SYSTEM FIO_Sorting_Station
  (* Version 1.0, 2022-03-11, Maximilian Scharf *)
  APPLICATION Sorting_Station
    (* Group __Group01: Human Machine Interface *)
    (* Group __Group02: Sensors *)
    (* Group __Group03: Factory IO data *)
    (* Group __Group04: Aktuatoren *)
    (* Group __Group05: Human Machine Interface *)
    (* Group __Group07: Factory IO data *)
    (* Group __Group09: Counter Ticker *)
    FBS
      E_R_TRIG : E_R_TRIG;
      BOOL2BOOL : BOOL2BOOL; {SET_ATTRIBUTE(GroupName, __Group02)}
      BOOL2BOOL_1 : BOOL2BOOL; {SET_ATTRIBUTE(GroupName, __Group01)}
      BOOL2BOOL_2 : BOOL2BOOL; {SET_ATTRIBUTE(GroupName, __Group01)}
      BOOL2BOOL_3 : BOOL2BOOL; {SET_ATTRIBUTE(GroupName, __Group01)}
      BOOL2BOOL_4 : BOOL2BOOL; {SET_ATTRIBUTE(GroupName, __Group01)}
      BOOL2BOOL_5 : BOOL2BOOL; {SET_ATTRIBUTE(GroupName, __Group01)}
      BOOL2BOOL_6 : BOOL2BOOL; {SET_ATTRIBUTE(GroupName, __Group01)}
      BOOL2BOOL_7 : BOOL2BOOL(IN := 0);
      BOOL2BOOL_8 : BOOL2BOOL(IN := 0);
      BOOL2BOOL_9 : BOOL2BOOL(IN := 0);
      BOOL2BOOL_10 : BOOL2BOOL(IN := 0);
      BOOL2BOOL_11 : BOOL2BOOL(IN := 0);
      BOOL2BOOL_18 : BOOL2BOOL;
      E_R_TRIG_2 : E_R_TRIG;
      Is_running : E_RS;
      E_F_TRIG : E_F_TRIG;
      Is_running_NOT : F_NOT;
      UINT2UINT : F_DINT_TO_UINT; {SET_ATTRIBUTE(GroupName, __Group02)}
      E_R_TRIG_1 : E_R_TRIG;
      F_SEL : F_SEL(IN0 := UINT#1);
      UINT2UINT_1 : UINT2UINT;
      UINT2UINT_2 : UINT2UINT;
      BOOL2BOOL_12 : BOOL2BOOL;
      UINT2UINT_3 : UINT2UINT;
      BOOL2BOOL_13 : BOOL2BOOL;
      UINT2UINT_4 : UINT2UINT;
      BOOL2BOOL_14 : BOOL2BOOL;
      BOOL2BOOL_15 : BOOL2BOOL;
      UINT2UINT_5 : UINT2UINT;
      UINT2UINT_6 : UINT2UINT; {SET_ATTRIBUTE(GroupName, __Group09)}
      BOOL2BOOL_16 : BOOL2BOOL;
      BOOL2BOOL_17 : BOOL2BOOL;
      UINT2UINT_7 : UINT2UINT;
      UINT2UINT_8 : UINT2UINT;
      UINT2UINT_9 : UINT2UINT; {SET_ATTRIBUTE(GroupName, __Group09)}
      UINT2UINT_10 : UINT2UINT; {SET_ATTRIBUTE(GroupName, __Group09)}
      BOOL2BOOL_19 : BOOL2BOOL;
      E_R_TRIG_3 : E_R_TRIG;
      BOOL2BOOL_20 : BOOL2BOOL;
      E_R_TRIG_4 : E_R_TRIG;
      BOOL2BOOL_21 : BOOL2BOOL;
      E_R_TRIG_5 : E_R_TRIG;
    END_FBS
    SUBAPPS
      FIO : OPC_SUB_FIO(QI := 1); {SET_ATTRIBUTE(GroupName, __Group03)}
      UPC_PUB_FIO : OPC_PUB_FIO(QI := 1); {SET_ATTRIBUTE(GroupName, __Group07)}
      Start_Light : OPC_PUB_1_FixID(QI := 1, prefix := "FIO_Q_", var1 := "start_light"); {SET_ATTRIBUTE(GroupName, __Group05)}
      Reset_Light : OPC_PUB_1_FixID(QI := 1, prefix := "FIO_Q_", var1 := "reset_light"); {SET_ATTRIBUTE(GroupName, __Group05)}
      Stop_Light : OPC_PUB_1_FixID(QI := 1, prefix := "FIO_Q_", var1 := "stop_light"); {SET_ATTRIBUTE(GroupName, __Group05)}
      ENTRY_CONVEYOR : OPC_PUB_1_FixID(QI := 1, prefix := "FIO_Q_", var1 := "entry_conveyor"); {SET_ATTRIBUTE(GroupName, __Group04)}
      EXIT_CONVEYOR : OPC_PUB_1_FixID(QI := 1, prefix := "FIO_Q_", var1 := "exit_conveyor"); {SET_ATTRIBUTE(GroupName, __Group04)}
      At_Exit : OPC_SUB_1_FixID(QI := 1, prefix := "FIO_I_", var1 := "at_exit"); {SET_ATTRIBUTE(GroupName, __Group02)}
      Vison_Sensor : OPC_SUB_1_FixID(QI := 1, prefix := "FIO_I_", var1 := "vision_sensor"); {SET_ATTRIBUTE(GroupName, __Group02)}
      Stop : OPC_SUB_1_FixID(QI := 1, prefix := "FIO_I_", var1 := "Stop"); {SET_ATTRIBUTE(GroupName, __Group01)}
      Reset : OPC_SUB_1_FixID(QI := 1, prefix := "FIO_I_", var1 := "reset"); {SET_ATTRIBUTE(GroupName, __Group01)}
      Emergency_Stop : OPC_SUB_1_FixID(QI := 1, prefix := "FIO_I_", var1 := "emergency_stop"); {SET_ATTRIBUTE(GroupName, __Group01)}
      Auto : OPC_SUB_1_FixID(QI := 1, prefix := "FIO_I_", var1 := "auto"); {SET_ATTRIBUTE(GroupName, __Group01)}
      Manual : OPC_SUB_1_FixID(QI := 1, prefix := "FIO_I_", var1 := "Manual"); {SET_ATTRIBUTE(GroupName, __Group01)}
      Start : OPC_SUB_1_FixID(QI := 1, prefix := "FIO_I_", var1 := "start"); {SET_ATTRIBUTE(GroupName, __Group01)}
      STOP_BLADE : OPC_PUB_1_FixID(QI := 1, prefix := "FIO_Q_", var1 := "stop_blade"); {SET_ATTRIBUTE(GroupName, __Group04)}
      Sorter_1 : Sorter(Prefix := "FIO_Q_", CountVar := "counter_1", BeltVar := "sorter_1_belt", TurnVar := "sorter_1_turn"); {SET_ATTRIBUTE(GroupName, __Group04)}
      Sorter_2 : Sorter(Prefix := "FIO_Q_", CountVar := "counter_2", BeltVar := "sorter_2_belt", TurnVar := "sorter_2_turn"); {SET_ATTRIBUTE(GroupName, __Group04)}
      Sorter_3 : Sorter(Prefix := "FIO_Q_", CountVar := "counter_3", BeltVar := "sorter_3_belt", TurnVar := "sorter_3_turn"); {SET_ATTRIBUTE(GroupName, __Group04)}
      OPC_PUB_1_FixID : OPC_PUB_1_FixID(QI := 1, prefix := "CON_", var1 := "sorter_1");
      OPC_PUB_EX_1 : OPC_PUB_EX_1(QI := 1, prefix := "FIO_Q_", var1 := "sorter_1_belt", server := WSTRING#"localhost:4840");
      OPC_PUB_EX_2 : OPC_PUB_EX_1(QI := 1, prefix := "FIO_Q_", var1 := "sorter_1_turn", server := WSTRING#"localhost:4840");
      OPC_SUB_EX_4 : OPC_SUB_EX_1(QI := 1, prefix := "CON_", var1 := "sorter_1", server := WSTRING#"localhost:4840");
      OPC_SUB_EX_5 : OPC_SUB_EX_1(QI := 1, prefix := "CON_", var1 := "sorter_2", server := WSTRING#"localhost:4840");
      OPC_PUB_EX_3 : OPC_PUB_EX_1(QI := 1, prefix := "FIO_Q_", var1 := "sorter_2_belt", server := WSTRING#"localhost:4840");
      OPC_PUB_EX_4 : OPC_PUB_EX_1(QI := 1, prefix := "FIO_Q_", var1 := "sorter_2_turn", server := WSTRING#"localhost:4840");
      OPC_PUB_EX_5 : OPC_PUB_EX_1(QI := 1, prefix := "FIO_Q_", var1 := "sorter_3_belt", server := WSTRING#"localhost:4840");
      OPC_SUB_EX_6 : OPC_SUB_EX_1(QI := 1, prefix := "CON_", var1 := "sorter_3", server := WSTRING#"localhost:4840");
      OPC_PUB_EX_6 : OPC_PUB_EX_1(QI := 1, prefix := "FIO_Q_", var1 := "sorter_3_turn", server := WSTRING#"localhost:4840");
      OPC_PUB_1_FixID_1 : OPC_PUB_1_FixID(QI := 1, prefix := "CON_", var1 := "sorter_2");
      OPC_PUB_1_FixID_2 : OPC_PUB_1_FixID(QI := 1, prefix := "CON_", var1 := "sorter_3");
      SorterLogic : SorterLogic(PackageNum := UINT#1);
      SorterLogic_3 : SorterLogic(PackageNum := UINT#2);
      SorterLogic_1 : SorterLogic(PackageNum := UINT#3);
      OPC_SUB_EX_7 : OPC_SUB_EX_1(QI := 1, prefix := "FIO_I_", var1 := "at_exit", server := WSTRING#"localhost:4840");
      OPC_SUB_1_FixID : OPC_SUB_1_FixID(QI := 1, prefix := "CON_", var1 := "C1"); {SET_ATTRIBUTE(GroupName, __Group09)}
      OPC_PUB_EX_7 : OPC_PUB_EX_1(QI := 1, prefix := "CON_", var1 := "C1", server := WSTRING#"localhost:4840");
      OPC_SUB_EX_8 : OPC_SUB_EX_1(QI := 1, prefix := "FIO_I_", var1 := "at_exit", server := WSTRING#"localhost:4840");
      OPC_SUB_EX_9 : OPC_SUB_EX_1(QI := 1, prefix := "FIO_I_", var1 := "at_exit", server := WSTRING#"localhost:4840");
      OPC_PUB_EX_8 : OPC_PUB_EX_1(QI := 1, prefix := "CON_", var1 := "C2", server := WSTRING#"localhost:4840");
      OPC_PUB_EX_9 : OPC_PUB_EX_1(QI := 1, prefix := "CON_", var1 := "C3", server := WSTRING#"localhost:4840");
      OPC_SUB_1_FixID_1 : OPC_SUB_1_FixID(QI := 1, prefix := "CON_", var1 := "C2"); {SET_ATTRIBUTE(GroupName, __Group09)}
      OPC_SUB_1_FixID_2 : OPC_SUB_1_FixID(QI := 1, prefix := "CON_", var1 := "C3"); {SET_ATTRIBUTE(GroupName, __Group09)}
      OPC_SUB_EX_1 : OPC_SUB_EX_1(QI := 1, prefix := "FIO_I_", var1 := "reset", server := WSTRING#"localhost:4840");
      OPC_SUB_EX_2 : OPC_SUB_EX_1(QI := 1, prefix := "FIO_I_", var1 := "reset", server := WSTRING#"localhost:4840");
      OPC_SUB_EX_3 : OPC_SUB_EX_1(QI := 1, prefix := "FIO_I_", var1 := "reset", server := WSTRING#"localhost:4840");
    END_SUBAPPS
    EVENT_CONNECTIONS
      BOOL2BOOL.CNF TO E_R_TRIG.EI;
      FIO.INITO TO UPC_PUB_FIO.INIT;
      At_Exit.IND TO BOOL2BOOL.REQ;
      Reset.IND TO BOOL2BOOL_1.REQ;
      Stop.IND TO BOOL2BOOL_3.REQ;
      Emergency_Stop.IND TO BOOL2BOOL_4.REQ;
      Auto.IND TO BOOL2BOOL_5.REQ;
      Manual.IND TO BOOL2BOOL_6.REQ;
      BOOL2BOOL_7.CNF TO Start_Light.REQ;
      BOOL2BOOL_8.CNF TO Reset_Light.REQ;
      BOOL2BOOL_9.CNF TO Stop_Light.REQ;
      BOOL2BOOL_10.CNF TO ENTRY_CONVEYOR.REQ;
      BOOL2BOOL_11.CNF TO EXIT_CONVEYOR.REQ;
      Start.IND TO BOOL2BOOL_2.REQ;
      BOOL2BOOL_18.CNF TO STOP_BLADE.REQ;
      BOOL2BOOL_2.CNF TO E_R_TRIG_2.EI;
      E_R_TRIG_2.EO TO Is_running.S;
      Is_running.EO TO BOOL2BOOL_7.REQ;
      Is_running.EO TO BOOL2BOOL_10.REQ;
      Is_running.EO TO BOOL2BOOL_11.REQ;
      BOOL2BOOL_3.CNF TO E_F_TRIG.EI;
      E_F_TRIG.EO TO Is_running.R;
      Is_running.EO TO Is_running_NOT.REQ;
      Is_running_NOT.CNF TO BOOL2BOOL_9.REQ;
      Is_running_NOT.CNF TO BOOL2BOOL_18.REQ;
      Vison_Sensor.IND TO UINT2UINT.REQ;
      BOOL2BOOL_1.CNF TO E_R_TRIG_1.EI;
      OPC_PUB_EX_1.INITO TO OPC_PUB_EX_2.INIT;
      OPC_SUB_EX_4.INITO TO OPC_PUB_EX_1.INIT;
      OPC_SUB_EX_5.INITO TO OPC_PUB_EX_3.INIT;
      OPC_PUB_EX_3.INITO TO OPC_PUB_EX_4.INIT;
      OPC_SUB_EX_6.INITO TO OPC_PUB_EX_5.INIT;
      OPC_PUB_EX_5.INITO TO OPC_PUB_EX_6.INIT;
      Is_running.EO TO F_SEL.REQ;
      UINT2UINT.CNF TO F_SEL.REQ;
      F_SEL.CNF TO UINT2UINT_1.REQ;
      UINT2UINT_1.CNF TO OPC_PUB_1_FixID.REQ;
      UINT2UINT_1.CNF TO OPC_PUB_1_FixID_1.REQ;
      UINT2UINT_1.CNF TO OPC_PUB_1_FixID_2.REQ;
      OPC_SUB_EX_4.IND TO UINT2UINT_2.REQ;
      UINT2UINT_2.CNF TO SorterLogic.IND;
      SorterLogic.CNF TO BOOL2BOOL_12.REQ;
      BOOL2BOOL_12.CNF TO OPC_PUB_EX_1.REQ;
      BOOL2BOOL_12.CNF TO OPC_PUB_EX_2.REQ;
      OPC_SUB_EX_5.IND TO UINT2UINT_3.REQ;
      UINT2UINT_3.CNF TO SorterLogic_3.IND;
      SorterLogic_3.CNF TO BOOL2BOOL_13.REQ;
      BOOL2BOOL_13.CNF TO OPC_PUB_EX_3.REQ;
      BOOL2BOOL_13.CNF TO OPC_PUB_EX_4.REQ;
      OPC_SUB_EX_6.IND TO UINT2UINT_4.REQ;
      UINT2UINT_4.CNF TO SorterLogic_1.IND;
      SorterLogic_1.CNF TO BOOL2BOOL_14.REQ;
      BOOL2BOOL_14.CNF TO OPC_PUB_EX_5.REQ;
      BOOL2BOOL_14.CNF TO OPC_PUB_EX_6.REQ;
      OPC_SUB_EX_4.INITO TO OPC_SUB_EX_7.INIT;
      UPC_PUB_FIO.INITO TO OPC_SUB_1_FixID.INIT;
      OPC_PUB_EX_2.INITO TO OPC_PUB_EX_7.INIT;
      OPC_SUB_EX_7.IND TO BOOL2BOOL_15.REQ;
      BOOL2BOOL_15.CNF TO SorterLogic.C;
      SorterLogic.CNT TO UINT2UINT_5.REQ;
      UINT2UINT_5.CNF TO OPC_PUB_EX_7.REQ;
      OPC_SUB_1_FixID.IND TO UINT2UINT_6.REQ;
      UINT2UINT_6.CNF TO Sorter_1.CNT;
      OPC_SUB_EX_5.INITO TO OPC_SUB_EX_8.INIT;
      OPC_SUB_EX_8.IND TO BOOL2BOOL_16.REQ;
      BOOL2BOOL_16.CNF TO SorterLogic_3.C;
      OPC_SUB_EX_6.INITO TO OPC_SUB_EX_9.INIT;
      OPC_SUB_EX_9.IND TO BOOL2BOOL_17.REQ;
      BOOL2BOOL_17.CNF TO SorterLogic_1.C;
      SorterLogic_3.CNT TO UINT2UINT_7.REQ;
      OPC_PUB_EX_4.INITO TO OPC_PUB_EX_8.INIT;
      UINT2UINT_7.CNF TO OPC_PUB_EX_8.REQ;
      SorterLogic_1.CNT TO UINT2UINT_8.REQ;
      OPC_PUB_EX_6.CNF TO OPC_PUB_EX_9.INIT;
      UINT2UINT_8.CNF TO OPC_PUB_EX_9.REQ;
      OPC_SUB_1_FixID.INITO TO OPC_SUB_1_FixID_1.INIT;
      OPC_SUB_1_FixID_1.IND TO UINT2UINT_9.REQ;
      UINT2UINT_9.CNF TO Sorter_2.CNT;
      OPC_SUB_1_FixID_1.INITO TO OPC_SUB_1_FixID_2.INIT;
      OPC_SUB_1_FixID_2.IND TO UINT2UINT_10.REQ;
      UINT2UINT_10.CNF TO Sorter_3.CNT;
      OPC_SUB_EX_1.IND TO BOOL2BOOL_19.REQ;
      BOOL2BOOL_19.CNF TO E_R_TRIG_3.EI;
      BOOL2BOOL_20.CNF TO E_R_TRIG_4.EI;
      OPC_SUB_EX_2.IND TO BOOL2BOOL_20.REQ;
      E_R_TRIG_4.EO TO SorterLogic_3.ResetC;
      OPC_SUB_EX_8.INITO TO OPC_SUB_EX_2.INIT;
      BOOL2BOOL_21.CNF TO E_R_TRIG_5.EI;
      OPC_SUB_EX_3.IND TO BOOL2BOOL_21.REQ;
      OPC_SUB_EX_9.INITO TO OPC_SUB_EX_3.INIT;
      E_R_TRIG_5.EO TO SorterLogic_1.ResetC;
      E_R_TRIG_3.EO TO SorterLogic.ResetC;
      OPC_SUB_EX_7.INITO TO OPC_SUB_EX_1.INIT;
    END_CONNECTIONS
    DATA_CONNECTIONS
      BOOL2BOOL.OUT TO E_R_TRIG.QI;
      At_Exit.value TO BOOL2BOOL.IN;
      Reset.value TO BOOL2BOOL_1.IN;
      Stop.value TO BOOL2BOOL_3.IN;
      Emergency_Stop.value TO BOOL2BOOL_4.IN;
      Auto.value TO BOOL2BOOL_5.IN;
      Manual.value TO BOOL2BOOL_6.IN;
      BOOL2BOOL_7.OUT TO Start_Light.value;
      BOOL2BOOL_8.OUT TO Reset_Light.value;
      BOOL2BOOL_9.OUT TO Stop_Light.value;
      BOOL2BOOL_10.OUT TO ENTRY_CONVEYOR.value;
      BOOL2BOOL_11.OUT TO EXIT_CONVEYOR.value;
      Start.value TO BOOL2BOOL_2.IN;
      BOOL2BOOL_18.OUT TO STOP_BLADE.value;
      BOOL2BOOL_2.OUT TO E_R_TRIG_2.QI;
      Is_running.Q TO BOOL2BOOL_7.IN;
      Is_running.Q TO BOOL2BOOL_10.IN;
      Is_running.Q TO BOOL2BOOL_11.IN;
      BOOL2BOOL_3.OUT TO E_F_TRIG.QI;
      Is_running.Q TO Is_running_NOT.IN;
      Is_running_NOT.OUT TO BOOL2BOOL_9.IN;
      Is_running_NOT.OUT TO BOOL2BOOL_18.IN;
      Vison_Sensor.value TO UINT2UINT.IN;
      BOOL2BOOL_1.OUT TO E_R_TRIG_1.QI;
      Is_running.Q TO F_SEL.G;
      UINT2UINT.OUT TO F_SEL.IN1;
      F_SEL.OUT TO UINT2UINT_1.IN;
      UINT2UINT_1.OUT TO OPC_PUB_1_FixID.value;
      UINT2UINT_1.OUT TO OPC_PUB_1_FixID_1.value;
      UINT2UINT_1.OUT TO OPC_PUB_1_FixID_2.value;
      OPC_SUB_EX_4.value TO UINT2UINT_2.IN;
      UINT2UINT_2.OUT TO SorterLogic.value;
      SorterLogic.OUT TO BOOL2BOOL_12.IN;
      BOOL2BOOL_12.OUT TO OPC_PUB_EX_1.value;
      BOOL2BOOL_12.OUT TO OPC_PUB_EX_2.value;
      OPC_SUB_EX_5.value TO UINT2UINT_3.IN;
      UINT2UINT_3.OUT TO SorterLogic_3.value;
      SorterLogic_3.OUT TO BOOL2BOOL_13.IN;
      BOOL2BOOL_13.OUT TO OPC_PUB_EX_3.value;
      BOOL2BOOL_13.OUT TO OPC_PUB_EX_4.value;
      OPC_SUB_EX_6.value TO UINT2UINT_4.IN;
      UINT2UINT_4.OUT TO SorterLogic_1.value;
      SorterLogic_1.OUT TO BOOL2BOOL_14.IN;
      BOOL2BOOL_14.OUT TO OPC_PUB_EX_5.value;
      BOOL2BOOL_14.OUT TO OPC_PUB_EX_6.value;
      OPC_SUB_EX_7.value TO BOOL2BOOL_15.IN;
      BOOL2BOOL_15.OUT TO SorterLogic.AtExit;
      SorterLogic.CV TO UINT2UINT_5.IN;
      UINT2UINT_5.OUT TO OPC_PUB_EX_7.value;
      OPC_SUB_1_FixID.value TO UINT2UINT_6.IN;
      UINT2UINT_6.OUT TO Sorter_1.Counter;
      OPC_SUB_EX_8.value TO BOOL2BOOL_16.IN;
      BOOL2BOOL_16.OUT TO SorterLogic_3.AtExit;
      OPC_SUB_EX_9.value TO BOOL2BOOL_17.IN;
      BOOL2BOOL_17.OUT TO SorterLogic_1.AtExit;
      SorterLogic_3.CV TO UINT2UINT_7.IN;
      UINT2UINT_7.OUT TO OPC_PUB_EX_8.value;
      SorterLogic_1.CV TO UINT2UINT_8.IN;
      UINT2UINT_8.OUT TO OPC_PUB_EX_9.value;
      OPC_SUB_1_FixID_1.value TO UINT2UINT_9.IN;
      UINT2UINT_9.OUT TO Sorter_2.Counter;
      OPC_SUB_1_FixID_2.value TO UINT2UINT_10.IN;
      UINT2UINT_10.OUT TO Sorter_3.Counter;
      OPC_SUB_EX_1.value TO BOOL2BOOL_19.IN;
      BOOL2BOOL_19.OUT TO E_R_TRIG_3.QI;
      BOOL2BOOL_20.OUT TO E_R_TRIG_4.QI;
      OPC_SUB_EX_2.value TO BOOL2BOOL_20.IN;
      BOOL2BOOL_21.OUT TO E_R_TRIG_5.QI;
      OPC_SUB_EX_3.value TO BOOL2BOOL_21.IN;
    END_CONNECTIONS
  END_APPLICATION
  DEVICE PLC : FORTE_PC(MGR_ID := "localhost:61600")
    {SET_ATTRIBUTE(Profile, DynamicTypeLoad)}
    {SET_ATTRIBUTE(FBType, GEN_E_MUX, F_LT, F_LWORD_TO_WORD, F_TAN, F_DINT_TO_UINT, F_BYTE_TO_DINT, F_ADD_DT_TIME, F_TIME_IN_US_TO_LREAL, F_INT_TO_UDINT, F_ADD_TOD_TIME, F_SUB_DT_DT, F_DT_TO_TOD, F_WSTRING_TO_REAL, F_UINT_TO_BCD_WORD, F_UDINT_TO_REAL, F_REAL_TO_UDINT, F_DWORD_TO_WORD, F_MUL, FB_CTUD_LINT, TEST_CONDITION, F_LE, GEN_SUBSCRIBE, F_LN, FB_CTD_DINT, GEN_OR, E_CYCLE, FB_F_TRIG, F_LREAL_TO_SINT, E_F_TRIG, F_LWORD_TO_UINT, E_RS, F_UINT_TO_WORD, F_WORD_TO_DINT, F_OR, F_WORD_TO_BYTE, F_TIME_IN_NS_TO_ULINT, FB_CTD_ULINT, FB_TOF, STEST_END, F_NE, FB_TON, F_STRING_TO_UINT, F_LWORD_TO_ULINT, F_INT_TO_STRING, F_INT_TO_BYTE, F_INT_TO_DINT, F_ULINT_TO_LINT, F_DWORD_TO_UINT, F_WSTRING_TO_ULINT, F_WSTRING_TO_LWORD, F_STRING_TO_DWORD, DWORD2DWORD, F_TIME_IN_NS_TO_LINT, F_DINT_TO_WSTRING, E_SELECT, F_LINT_TO_STRING, FB_CTUD, F_MULTIME, F_USINT_TO_INT, LocalizedText2LocalizedText, F_DWORD_TO_UDINT, F_UINT_TO_LWORD, F_SINT_TO_LWORD, GEN_F_MUX, USINT2USINT, F_LINT_TO_SINT, F_WORD_TO_USINT, F_DWORD_TO_INT, F_LREAL_TO_REAL, F_BOOL_TO_LINT, F_LEFT, FB_CTD, E_SR, F_UDINT_TO_BCD_DWORD, GEN_XOR, F_DINT_TO_WORD, F_SUB_TOD_TIME, E_RESTART, E_PERMIT, TIME2TIME, F_UINT_TO_SINT, F_XOR, F_STRING_TO_WORD, F_SEL, F_ULINT_TO_LREAL, F_SINT_TO_LREAL, F_DINT_TO_SINT, E_TimeOut, F_BYTE_TO_UDINT, F_REPLACE, F_LINT_TO_USINT, F_ABS, F_WORD_TO_LWORD, E_DELAY, GEN_ADD, F_INT_TO_WSTRING, F_STRING_TO_ULINT, F_USINT_TO_STRING, F_DINT_TO_USINT, F_STRING_TO_BOOL, F_DWORD_TO_WSTRING, F_INT_TO_REAL, F_DWORD_TO_STRING, E_CTU, F_TIME_TO_STRING, F_WSTRING_TO_BYTE, F_USINT_TO_WSTRING, F_WSTRING_TO_DINT, F_WSTRING_TO_DWORD, F_MOVE, F_WSTRING_TO_STRING, F_USINT_TO_LINT, F_DIV, F_WSTRING_TO_SINT, E_CTD, F_UINT_TO_DWORD, F_LWORD_TO_LINT, F_STRING_TO_TIME, FB_CTUD_DINT, F_ADD, F_BYTE_TO_LINT, F_TIME_IN_MS_TO_LREAL, F_LREAL_TO_UINT, F_ACOS, F_DWORD_TO_LINT, F_SHL, F_REAL_TO_ULINT, F_ULINT_TO_UINT, F_UDINT_TO_SINT, F_SHR, F_BOOL_TO_INT, UINT2UINT, F_WORD_TO_DWORD, F_INT_TO_LWORD, F_USINT_TO_UINT, F_LREAL_TO_WSTRING, F_INT_TO_ULINT, GEN_CSV_WRITER, F_LINT_TO_WORD, F_UINT_TO_LREAL, F_STRING_TO_SINT, F_SINT_TO_WORD, F_STRING_TO_WSTRING, STRING2STRING, F_LREAL_TO_DINT, F_SIN, F_UINT_TO_USINT, FB_CTU_LINT, F_DINT_TO_ULINT, F_REAL_TO_UINT, RMT_RES, F_ULINT_TO_WORD, F_INT_TO_LINT, E_D_FF, F_STRING_TO_USINT, FB_CTD_LINT, FB_R_TRIG, F_INT_TO_DWORD, F_WORD_TO_LINT, F_UDINT_TO_INT, REAL2REAL, F_LREAL_TO_STRING, F_WSTRING_TO_INT, F_LREAL_TO_USINT, F_DINT_TO_LWORD, DEV_MGR, F_SINT_TO_UINT, E_CTUD, E_RDELAY, F_SINT_TO_ULINT, F_LINT_TO_ULINT, F_RIGHT, F_SINT_TO_INT, F_LWORD_TO_WSTRING, SINT2SINT, FB_CTD_UDINT, F_LINT_TO_LWORD, F_LWORD_TO_UDINT, F_LWORD_TO_STRING, F_TRUNC, F_ULINT_TO_DWORD, F_TIME_IN_S_TO_LREAL, F_BOOL_TO_DWORD, E_TRAIN, OUT_ANY_CONSOLE, F_ULINT_TO_SINT, F_DINT_TO_LINT, F_BOOL_TO_USINT, F_UDINT_TO_DWORD, GEN_E_DEMUX, F_SQRT, F_BOOL_TO_DINT, F_BOOL_TO_BYTE, F_UINT_TO_INT, F_TIME_IN_S_TO_LINT, F_ULINT_TO_USINT, F_UINT_TO_REAL, F_LREAL_TO_LWORD, F_SINT_TO_LINT, F_MAX, F_LREAL_TO_INT, F_UDINT_TO_LWORD, INT2INT, F_BYTE_TO_ULINT, F_UDINT_TO_WORD, F_LINT_TO_UINT, F_TIME_IN_US_TO_ULINT, F_COS, F_TIME_IN_NS_TO_LREAL, F_REAL_TO_LINT, F_STRING_TO_LWORD, F_BYTE_TO_STRING, F_USINT_TO_WORD, E_REND, F_ASIN, F_REAL_TO_INT, F_BOOL_TO_LWORD, F_WORD_BCD_TO_UINT, F_BOOL_TO_SINT, F_BYTE_TO_INT, F_BOOL_TO_ULINT, EMB_RES, F_BYTE_TO_WORD, F_STRING_TO_INT, F_USINT_TO_LWORD, F_DWORD_TO_DINT, F_ULINT_TO_LWORD, GEN_APPEND_STRING, F_USINT_TO_ULINT, GEN_SUBL, F_DWORD_TO_BYTE, F_DIVTIME, F_ROL, F_LWORD_TO_DINT, F_WORD_TO_SINT, F_STRING_TO_REAL, F_LWORD_TO_BYTE, FB_CTU_DINT, GEN_AND, F_AND, F_ROR, GEN_CLIENT, F_ULINT_TO_WSTRING, F_SINT_TO_STRING, F_LREAL_TO_LINT, WSTRING2WSTRING, F_WORD_TO_INT, F_UINT_TO_BYTE, F_UDINT_TO_UINT, F_SINT_TO_UDINT, F_UINT_TO_DINT, F_UINT_TO_UDINT, F_UINT_TO_WSTRING, F_WSTRING_TO_UINT, F_DINT_TO_UDINT, E_SPLIT, F_DWORD_TO_LWORD, F_USINT_TO_SINT, F_ULINT_TO_BCD_LWORD, F_BYTE_BCD_TO_USINT, F_DWORD_TO_ULINT, F_BYTE_TO_SINT, F_BYTE_TO_WSTRING, GEN_ARRAY2ARRAY, F_DT_TO_DATE, GEN_STRUCT_DEMUX, F_LEN, GEN_STRUCT_MUX, F_INT_TO_WORD, FB_RANDOM, F_LINT_TO_UDINT, F_EXP, F_USINT_TO_DWORD, F_TIME_IN_MS_TO_ULINT, F_REAL_TO_SINT, F_INT_TO_USINT, F_UDINT_TO_WSTRING, F_EXPT, F_SUB, F_ULINT_TO_REAL, F_REAL_TO_LREAL, F_MID, F_BYTE_TO_UINT, F_BYTE_TO_DWORD, F_INT_TO_UINT, F_DWORD_TO_REAL, F_DINT_TO_BYTE, F_WORD_TO_STRING, F_REAL_TO_STRING, F_SUB_TOD_TOD, SET_AT_INDEX, F_MIN, F_LREAL_TO_ULINT, F_STRING_TO_BYTE, F_BYTE_TO_LWORD, F_STRING_TO_DINT, F_WORD_TO_WSTRING, BOOL2BOOL, F_LINT_TO_INT, F_WSTRING_TO_TIME, FB_CTU_UDINT, F_WSTRING_TO_BOOL, F_INSERT, F_SUB_DT_TIME, F_FIND, F_UDINT_TO_ULINT, F_WORD_TO_UDINT, F_DINT_TO_DWORD, F_WSTRING_TO_USINT, GEN_VALUES2ARRAY, GEN_ARRAY2VALUES, F_WSTRING_TO_WORD, F_DINT_TO_STRING, F_WORD_TO_UINT, F_TIME_IN_US_TO_LINT, F_LINT_TO_DWORD, F_CONCAT, FB_CTUD_ULINT, F_UDINT_TO_LINT, F_SUB_DATE_DATE, F_LWORD_TO_LREAL, F_LWORD_TO_INT, WORD2WORD, E_STOPWATCH, F_LIMIT, F_TIME_IN_S_TO_ULINT, F_LWORD_TO_USINT, F_REAL_TO_DINT, F_DWORD_TO_USINT, E_MERGE, F_SINT_TO_DWORD, E_DEMUX, F_BOOL_TO_UDINT, BYTE2BYTE, FB_TP, F_USINT_TO_BCD_BYTE, F_SINT_TO_DINT, F_UINT_TO_LINT, F_SINT_TO_BYTE, F_ATAN, F_LINT_TO_BYTE, F_BYTE_TO_USINT, F_ULINT_TO_UDINT, FB_SR, F_NOT, F_DINT_TO_INT, F_LINT_TO_DINT, F_DELETE, FB_CTU, GEN_SERVER, GEN_PUBL, F_UDINT_TO_LREAL, F_BOOL_TO_UINT, F_UINT_TO_STRING, E_R_TRIG, F_GE, F_LWORD_BCD_TO_ULINT, F_UDINT_TO_STRING, F_REAL_TO_WSTRING, FB_RS, F_MUX_2, F_LINT_TO_WSTRING, F_USINT_TO_UDINT, F_UINT_TO_ULINT, F_EQ, E_T_FF, F_USINT_TO_REAL, LREAL2LREAL, F_STRING_TO_LREAL, F_ULINT_TO_STRING, F_MOD, E_RTimeOut, F_ULINT_TO_DINT, F_ULINT_TO_BYTE, F_WSTRING_TO_UDINT, F_TIME_TO_WSTRING, GET_STRUCT_VALUE, GEN_PUBLISH, F_REAL_TO_DWORD, F_DWORD_BCD_TO_UDINT, F_INT_TO_LREAL, F_SINT_TO_WSTRING, F_LWORD_TO_SINT, F_GT, F_LINT_TO_REAL, F_TIME_IN_MS_TO_LINT, F_SINT_TO_REAL, F_LOG, F_ULINT_TO_INT, F_DWORD_TO_SINT, F_BOOL_TO_WORD, F_REAL_TO_USINT, E_SWITCH, F_LINT_TO_LREAL, F_STRING_TO_LINT, F_SINT_TO_USINT, F_DINT_TO_REAL, DINT2DINT, F_WORD_TO_ULINT, F_INT_TO_SINT, F_CONCAT_DATE_TOD, F_WSTRING_TO_LREAL, GET_AT_INDEX, F_USINT_TO_LREAL, F_BOOL_TO_WSTRING, FB_CTU_ULINT, F_DINT_TO_LREAL, UDINT2UDINT, F_USINT_TO_BYTE, F_BOOL_TO_STRING, F_LWORD_TO_DWORD, F_LREAL_TO_UDINT, F_STRING_TO_UDINT, F_UDINT_TO_DINT, F_UDINT_TO_BYTE, F_WSTRING_TO_LINT, F_USINT_TO_DINT)} (* created during deployment *)
    RESOURCE CPU1 : EMB_RES
      FBS
        E_R_TRIG : E_R_TRIG;
        BOOL2BOOL : BOOL2BOOL;
        BOOL2BOOL_1 : BOOL2BOOL;
        BOOL2BOOL_2 : BOOL2BOOL;
        BOOL2BOOL_3 : BOOL2BOOL;
        BOOL2BOOL_4 : BOOL2BOOL;
        BOOL2BOOL_5 : BOOL2BOOL;
        BOOL2BOOL_6 : BOOL2BOOL;
        BOOL2BOOL_7 : BOOL2BOOL(IN := 0);
        BOOL2BOOL_8 : BOOL2BOOL(IN := 0);
        BOOL2BOOL_9 : BOOL2BOOL(IN := 0);
        BOOL2BOOL_10 : BOOL2BOOL(IN := 0);
        BOOL2BOOL_11 : BOOL2BOOL(IN := 0);
        BOOL2BOOL_18 : BOOL2BOOL;
        E_R_TRIG_2 : E_R_TRIG;
        Is_running : E_RS;
        E_F_TRIG : E_F_TRIG;
        Is_running_NOT : F_NOT;
        UINT2UINT : F_DINT_TO_UINT;
        E_R_TRIG_1 : E_R_TRIG;
        F_SEL : F_SEL(IN0 := UINT#1);
        UINT2UINT_1 : UINT2UINT;
        UINT2UINT_6 : UINT2UINT;
        UINT2UINT_9 : UINT2UINT;
        UINT2UINT_10 : UINT2UINT;
      END_FBS
      SUBAPPS
        FIO : OPC_SUB_FIO(QI := 1);
        UPC_PUB_FIO : OPC_PUB_FIO(QI := 1);
        Start_Light : OPC_PUB_1_FixID(QI := 1, prefix := "FIO_Q_", var1 := "start_light");
        Reset_Light : OPC_PUB_1_FixID(QI := 1, prefix := "FIO_Q_", var1 := "reset_light");
        Stop_Light : OPC_PUB_1_FixID(QI := 1, prefix := "FIO_Q_", var1 := "stop_light");
        ENTRY_CONVEYOR : OPC_PUB_1_FixID(QI := 1, prefix := "FIO_Q_", var1 := "entry_conveyor");
        EXIT_CONVEYOR : OPC_PUB_1_FixID(QI := 1, prefix := "FIO_Q_", var1 := "exit_conveyor");
        At_Exit : OPC_SUB_1_FixID(QI := 1, prefix := "FIO_I_", var1 := "at_exit");
        Vison_Sensor : OPC_SUB_1_FixID(QI := 1, prefix := "FIO_I_", var1 := "vision_sensor");
        Stop : OPC_SUB_1_FixID(QI := 1, prefix := "FIO_I_", var1 := "Stop");
        Reset : OPC_SUB_1_FixID(QI := 1, prefix := "FIO_I_", var1 := "reset");
        Emergency_Stop : OPC_SUB_1_FixID(QI := 1, prefix := "FIO_I_", var1 := "emergency_stop");
        Auto : OPC_SUB_1_FixID(QI := 1, prefix := "FIO_I_", var1 := "auto");
        Manual : OPC_SUB_1_FixID(QI := 1, prefix := "FIO_I_", var1 := "Manual");
        Start : OPC_SUB_1_FixID(QI := 1, prefix := "FIO_I_", var1 := "start");
        STOP_BLADE : OPC_PUB_1_FixID(QI := 1, prefix := "FIO_Q_", var1 := "stop_blade");
        Sorter_1 : Sorter(Prefix := "FIO_Q_", CountVar := "counter_1", BeltVar := "sorter_1_belt", TurnVar := "sorter_1_turn");
        Sorter_2 : Sorter(Prefix := "FIO_Q_", CountVar := "counter_2", BeltVar := "sorter_2_belt", TurnVar := "sorter_2_turn");
        Sorter_3 : Sorter(Prefix := "FIO_Q_", CountVar := "counter_3", BeltVar := "sorter_3_belt", TurnVar := "sorter_3_turn");
        OPC_PUB_1_FixID : OPC_PUB_1_FixID(QI := 1, prefix := "CON_", var1 := "sorter_1");
        OPC_PUB_1_FixID_1 : OPC_PUB_1_FixID(QI := 1, prefix := "CON_", var1 := "sorter_2");
        OPC_PUB_1_FixID_2 : OPC_PUB_1_FixID(QI := 1, prefix := "CON_", var1 := "sorter_3");
        OPC_SUB_1_FixID : OPC_SUB_1_FixID(QI := 1, prefix := "CON_", var1 := "C1");
        OPC_SUB_1_FixID_1 : OPC_SUB_1_FixID(QI := 1, prefix := "CON_", var1 := "C2");
        OPC_SUB_1_FixID_2 : OPC_SUB_1_FixID(QI := 1, prefix := "CON_", var1 := "C3");
      END_SUBAPPS
      EVENT_CONNECTIONS
        START.COLD TO FIO.INIT;
        BOOL2BOOL.CNF TO E_R_TRIG.EI;
        FIO.INITO TO UPC_PUB_FIO.INIT;
        START.COLD TO Start_Light.INIT;
        START.COLD TO Reset_Light.INIT;
        START.COLD TO Stop_Light.INIT;
        START.COLD TO ENTRY_CONVEYOR.INIT;
        START.COLD TO EXIT_CONVEYOR.INIT;
        At_Exit.IND TO BOOL2BOOL.REQ;
        START.COLD TO At_Exit.INIT;
        START.COLD TO Vison_Sensor.INIT;
        START.COLD TO Stop.INIT;
        Reset.IND TO BOOL2BOOL_1.REQ;
        START.COLD TO Reset.INIT;
        START.COLD TO Emergency_Stop.INIT;
        START.COLD TO Auto.INIT;
        START.COLD TO Manual.INIT;
        Stop.IND TO BOOL2BOOL_3.REQ;
        Emergency_Stop.IND TO BOOL2BOOL_4.REQ;
        Auto.IND TO BOOL2BOOL_5.REQ;
        Manual.IND TO BOOL2BOOL_6.REQ;
        BOOL2BOOL_7.CNF TO Start_Light.REQ;
        BOOL2BOOL_8.CNF TO Reset_Light.REQ;
        BOOL2BOOL_9.CNF TO Stop_Light.REQ;
        BOOL2BOOL_10.CNF TO ENTRY_CONVEYOR.REQ;
        BOOL2BOOL_11.CNF TO EXIT_CONVEYOR.REQ;
        Start.IND TO BOOL2BOOL_2.REQ;
        START.COLD TO Start.INIT;
        START.COLD TO STOP_BLADE.INIT;
        BOOL2BOOL_18.CNF TO STOP_BLADE.REQ;
        BOOL2BOOL_2.CNF TO E_R_TRIG_2.EI;
        E_R_TRIG_2.EO TO Is_running.S;
        Is_running.EO TO BOOL2BOOL_7.REQ;
        Is_running.EO TO BOOL2BOOL_10.REQ;
        Is_running.EO TO BOOL2BOOL_11.REQ;
        BOOL2BOOL_3.CNF TO E_F_TRIG.EI;
        E_F_TRIG.EO TO Is_running.R;
        Is_running.EO TO Is_running_NOT.REQ;
        Is_running_NOT.CNF TO BOOL2BOOL_9.REQ;
        Is_running_NOT.CNF TO BOOL2BOOL_18.REQ;
        Vison_Sensor.IND TO UINT2UINT.REQ;
        BOOL2BOOL_1.CNF TO E_R_TRIG_1.EI;
        START.COLD TO Sorter_1.INIT;
        START.COLD TO Sorter_2.INIT;
        START.COLD TO Sorter_3.INIT;
        START.COLD TO OPC_PUB_1_FixID.INIT;
        START.COLD TO OPC_PUB_1_FixID_1.INIT;
        START.COLD TO OPC_PUB_1_FixID_2.INIT;
        Is_running.EO TO F_SEL.REQ;
        UINT2UINT.CNF TO F_SEL.REQ;
        F_SEL.CNF TO UINT2UINT_1.REQ;
        UINT2UINT_1.CNF TO OPC_PUB_1_FixID.REQ;
        UINT2UINT_1.CNF TO OPC_PUB_1_FixID_1.REQ;
        UINT2UINT_1.CNF TO OPC_PUB_1_FixID_2.REQ;
        UPC_PUB_FIO.INITO TO OPC_SUB_1_FixID.INIT;
        OPC_SUB_1_FixID.IND TO UINT2UINT_6.REQ;
        UINT2UINT_6.CNF TO Sorter_1.CNT;
        OPC_SUB_1_FixID.INITO TO OPC_SUB_1_FixID_1.INIT;
        OPC_SUB_1_FixID_1.IND TO UINT2UINT_9.REQ;
        UINT2UINT_9.CNF TO Sorter_2.CNT;
        OPC_SUB_1_FixID_1.INITO TO OPC_SUB_1_FixID_2.INIT;
        OPC_SUB_1_FixID_2.IND TO UINT2UINT_10.REQ;
        UINT2UINT_10.CNF TO Sorter_3.CNT;
      END_CONNECTIONS
      DATA_CONNECTIONS
        BOOL2BOOL.OUT TO E_R_TRIG.QI;
        At_Exit.value TO BOOL2BOOL.IN;
        Reset.value TO BOOL2BOOL_1.IN;
        Stop.value TO BOOL2BOOL_3.IN;
        Emergency_Stop.value TO BOOL2BOOL_4.IN;
        Auto.value TO BOOL2BOOL_5.IN;
        Manual.value TO BOOL2BOOL_6.IN;
        BOOL2BOOL_7.OUT TO Start_Light.value;
        BOOL2BOOL_8.OUT TO Reset_Light.value;
        BOOL2BOOL_9.OUT TO Stop_Light.value;
        BOOL2BOOL_10.OUT TO ENTRY_CONVEYOR.value;
        BOOL2BOOL_11.OUT TO EXIT_CONVEYOR.value;
        Start.value TO BOOL2BOOL_2.IN;
        BOOL2BOOL_18.OUT TO STOP_BLADE.value;
        BOOL2BOOL_2.OUT TO E_R_TRIG_2.QI;
        Is_running.Q TO BOOL2BOOL_7.IN;
        Is_running.Q TO BOOL2BOOL_10.IN;
        Is_running.Q TO BOOL2BOOL_11.IN;
        BOOL2BOOL_3.OUT TO E_F_TRIG.QI;
        Is_running.Q TO Is_running_NOT.IN;
        Is_running_NOT.OUT TO BOOL2BOOL_9.IN;
        Is_running_NOT.OUT TO BOOL2BOOL_18.IN;
        Vison_Sensor.value TO UINT2UINT.IN;
        BOOL2BOOL_1.OUT TO E_R_TRIG_1.QI;
        Is_running.Q TO F_SEL.G;
        UINT2UINT.OUT TO F_SEL.IN1;
        F_SEL.OUT TO UINT2UINT_1.IN;
        UINT2UINT_1.OUT TO OPC_PUB_1_FixID.value;
        UINT2UINT_1.OUT TO OPC_PUB_1_FixID_1.value;
        UINT2UINT_1.OUT TO OPC_PUB_1_FixID_2.value;
        OPC_SUB_1_FixID.value TO UINT2UINT_6.IN;
        UINT2UINT_6.OUT TO Sorter_1.Counter;
        OPC_SUB_1_FixID_1.value TO UINT2UINT_9.IN;
        UINT2UINT_9.OUT TO Sorter_2.Counter;
        OPC_SUB_1_FixID_2.value TO UINT2UINT_10.IN;
        UINT2UINT_10.OUT TO Sorter_3.Counter;
      END_CONNECTIONS
    END_RESOURCE
    RESOURCE CPU2 : EMB_RES
    END_RESOURCE
  END_DEVICE
  DEVICE SorterUnit1 : FORTE_PC(MGR_ID := "localhost:61601")
    {SET_ATTRIBUTE(Profile, HOLOBLOC)}
    RESOURCE EMB_RES : EMB_RES
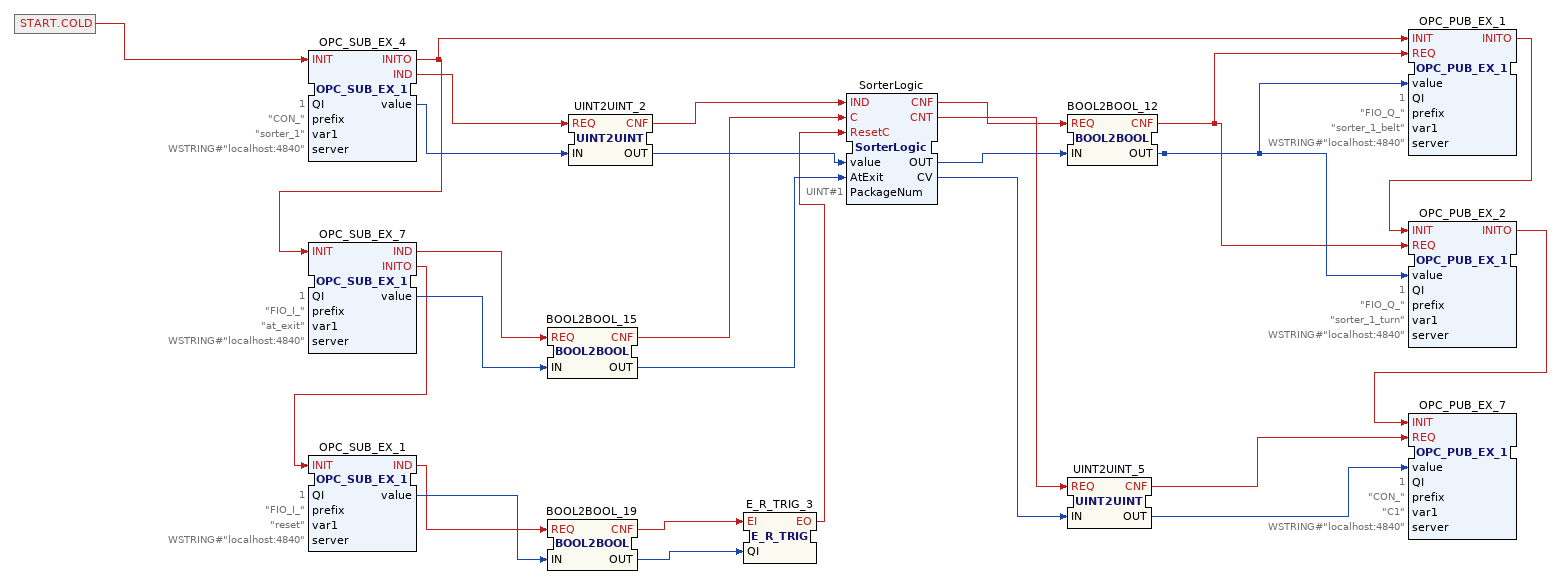
      FBS
        UINT2UINT_2 : UINT2UINT;
        BOOL2BOOL_12 : BOOL2BOOL;
        BOOL2BOOL_15 : BOOL2BOOL;
        UINT2UINT_5 : UINT2UINT;
        BOOL2BOOL_19 : BOOL2BOOL;
        E_R_TRIG_3 : E_R_TRIG;
      END_FBS
      SUBAPPS
        OPC_PUB_EX_1 : OPC_PUB_EX_1(QI := 1, prefix := "FIO_Q_", var1 := "sorter_1_belt", server := WSTRING#"localhost:4840");
        OPC_PUB_EX_2 : OPC_PUB_EX_1(QI := 1, prefix := "FIO_Q_", var1 := "sorter_1_turn", server := WSTRING#"localhost:4840");
        OPC_SUB_EX_4 : OPC_SUB_EX_1(QI := 1, prefix := "CON_", var1 := "sorter_1", server := WSTRING#"localhost:4840");
        SorterLogic : SorterLogic(PackageNum := UINT#1);
        OPC_SUB_EX_7 : OPC_SUB_EX_1(QI := 1, prefix := "FIO_I_", var1 := "at_exit", server := WSTRING#"localhost:4840");
        OPC_PUB_EX_7 : OPC_PUB_EX_1(QI := 1, prefix := "CON_", var1 := "C1", server := WSTRING#"localhost:4840");
        OPC_SUB_EX_1 : OPC_SUB_EX_1(QI := 1, prefix := "FIO_I_", var1 := "reset", server := WSTRING#"localhost:4840");
      END_SUBAPPS
      EVENT_CONNECTIONS
        OPC_PUB_EX_1.INITO TO OPC_PUB_EX_2.INIT;
        OPC_SUB_EX_4.INITO TO OPC_PUB_EX_1.INIT;
        START.COLD TO OPC_SUB_EX_4.INIT;
        OPC_SUB_EX_4.IND TO UINT2UINT_2.REQ;
        UINT2UINT_2.CNF TO SorterLogic.IND;
        SorterLogic.CNF TO BOOL2BOOL_12.REQ;
        BOOL2BOOL_12.CNF TO OPC_PUB_EX_1.REQ;
        BOOL2BOOL_12.CNF TO OPC_PUB_EX_2.REQ;
        OPC_SUB_EX_4.INITO TO OPC_SUB_EX_7.INIT;
        OPC_PUB_EX_2.INITO TO OPC_PUB_EX_7.INIT;
        OPC_SUB_EX_7.IND TO BOOL2BOOL_15.REQ;
        BOOL2BOOL_15.CNF TO SorterLogic.C;
        SorterLogic.CNT TO UINT2UINT_5.REQ;
        UINT2UINT_5.CNF TO OPC_PUB_EX_7.REQ;
        BOOL2BOOL_19.CNF TO E_R_TRIG_3.EI;
        OPC_SUB_EX_1.IND TO BOOL2BOOL_19.REQ;
        E_R_TRIG_3.EO TO SorterLogic.ResetC;
        OPC_SUB_EX_7.INITO TO OPC_SUB_EX_1.INIT;
      END_CONNECTIONS
      DATA_CONNECTIONS
        OPC_SUB_EX_4.value TO UINT2UINT_2.IN;
        UINT2UINT_2.OUT TO SorterLogic.value;
        SorterLogic.OUT TO BOOL2BOOL_12.IN;
        BOOL2BOOL_12.OUT TO OPC_PUB_EX_1.value;
        BOOL2BOOL_12.OUT TO OPC_PUB_EX_2.value;
        OPC_SUB_EX_7.value TO BOOL2BOOL_15.IN;
        BOOL2BOOL_15.OUT TO SorterLogic.AtExit;
        SorterLogic.CV TO UINT2UINT_5.IN;
        UINT2UINT_5.OUT TO OPC_PUB_EX_7.value;
        BOOL2BOOL_19.OUT TO E_R_TRIG_3.QI;
        OPC_SUB_EX_1.value TO BOOL2BOOL_19.IN;
      END_CONNECTIONS
    END_RESOURCE
  END_DEVICE
  DEVICE SorterUnit2 : FORTE_PC(MGR_ID := "localhost:61602")
    {SET_ATTRIBUTE(Profile, HOLOBLOC)}
    RESOURCE EMB_RES : EMB_RES
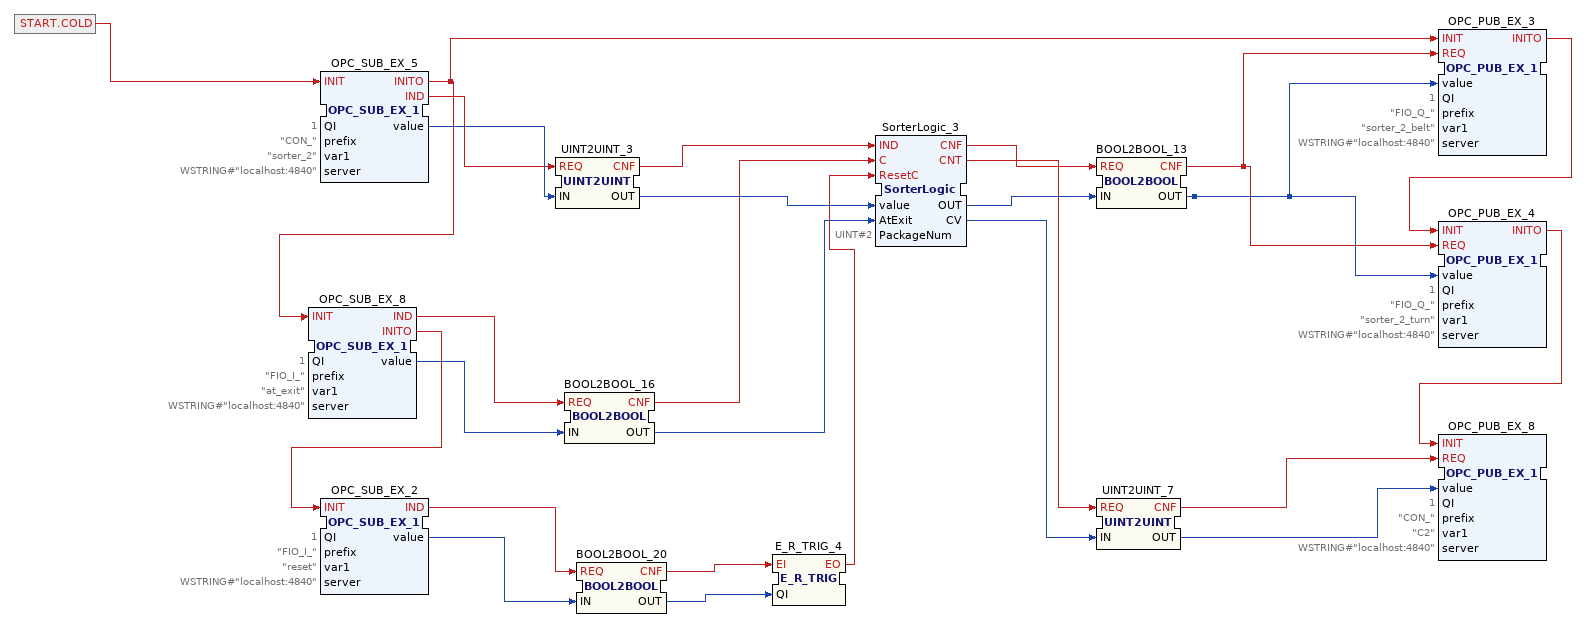
      FBS
        UINT2UINT_3 : UINT2UINT;
        BOOL2BOOL_13 : BOOL2BOOL;
        BOOL2BOOL_16 : BOOL2BOOL;
        UINT2UINT_7 : UINT2UINT;
        E_R_TRIG_4 : E_R_TRIG;
        BOOL2BOOL_20 : BOOL2BOOL;
      END_FBS
      SUBAPPS
        OPC_SUB_EX_5 : OPC_SUB_EX_1(QI := 1, prefix := "CON_", var1 := "sorter_2", server := WSTRING#"localhost:4840");
        OPC_PUB_EX_3 : OPC_PUB_EX_1(QI := 1, prefix := "FIO_Q_", var1 := "sorter_2_belt", server := WSTRING#"localhost:4840");
        OPC_PUB_EX_4 : OPC_PUB_EX_1(QI := 1, prefix := "FIO_Q_", var1 := "sorter_2_turn", server := WSTRING#"localhost:4840");
        SorterLogic_3 : SorterLogic(PackageNum := UINT#2);
        OPC_SUB_EX_8 : OPC_SUB_EX_1(QI := 1, prefix := "FIO_I_", var1 := "at_exit", server := WSTRING#"localhost:4840");
        OPC_PUB_EX_8 : OPC_PUB_EX_1(QI := 1, prefix := "CON_", var1 := "C2", server := WSTRING#"localhost:4840");
        OPC_SUB_EX_2 : OPC_SUB_EX_1(QI := 1, prefix := "FIO_I_", var1 := "reset", server := WSTRING#"localhost:4840");
      END_SUBAPPS
      EVENT_CONNECTIONS
        START.COLD TO OPC_SUB_EX_5.INIT;
        OPC_SUB_EX_5.INITO TO OPC_PUB_EX_3.INIT;
        OPC_PUB_EX_3.INITO TO OPC_PUB_EX_4.INIT;
        OPC_SUB_EX_5.IND TO UINT2UINT_3.REQ;
        UINT2UINT_3.CNF TO SorterLogic_3.IND;
        SorterLogic_3.CNF TO BOOL2BOOL_13.REQ;
        BOOL2BOOL_13.CNF TO OPC_PUB_EX_3.REQ;
        BOOL2BOOL_13.CNF TO OPC_PUB_EX_4.REQ;
        OPC_SUB_EX_5.INITO TO OPC_SUB_EX_8.INIT;
        OPC_SUB_EX_8.IND TO BOOL2BOOL_16.REQ;
        BOOL2BOOL_16.CNF TO SorterLogic_3.C;
        SorterLogic_3.CNT TO UINT2UINT_7.REQ;
        OPC_PUB_EX_4.INITO TO OPC_PUB_EX_8.INIT;
        UINT2UINT_7.CNF TO OPC_PUB_EX_8.REQ;
        OPC_SUB_EX_8.INITO TO OPC_SUB_EX_2.INIT;
        E_R_TRIG_4.EO TO SorterLogic_3.ResetC;
        OPC_SUB_EX_2.IND TO BOOL2BOOL_20.REQ;
        BOOL2BOOL_20.CNF TO E_R_TRIG_4.EI;
      END_CONNECTIONS
      DATA_CONNECTIONS
        OPC_SUB_EX_5.value TO UINT2UINT_3.IN;
        UINT2UINT_3.OUT TO SorterLogic_3.value;
        SorterLogic_3.OUT TO BOOL2BOOL_13.IN;
        BOOL2BOOL_13.OUT TO OPC_PUB_EX_3.value;
        BOOL2BOOL_13.OUT TO OPC_PUB_EX_4.value;
        OPC_SUB_EX_8.value TO BOOL2BOOL_16.IN;
        BOOL2BOOL_16.OUT TO SorterLogic_3.AtExit;
        SorterLogic_3.CV TO UINT2UINT_7.IN;
        UINT2UINT_7.OUT TO OPC_PUB_EX_8.value;
        OPC_SUB_EX_2.value TO BOOL2BOOL_20.IN;
        BOOL2BOOL_20.OUT TO E_R_TRIG_4.QI;
      END_CONNECTIONS
    END_RESOURCE
  END_DEVICE
  DEVICE SorterUnit3 : FORTE_PC(MGR_ID := "localhost:61603")
    {SET_ATTRIBUTE(Profile, HOLOBLOC)}
    RESOURCE EMB_RES : EMB_RES
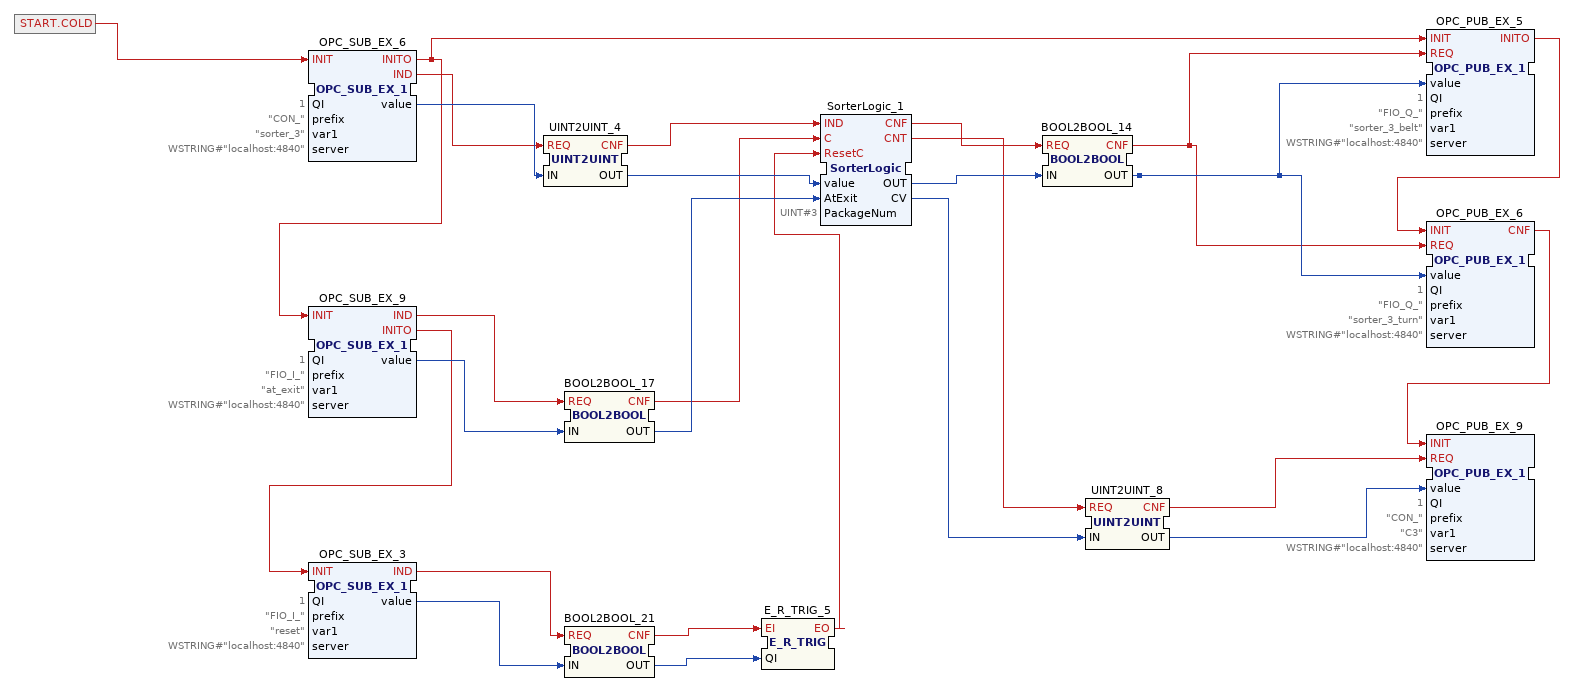
      FBS
        UINT2UINT_4 : UINT2UINT;
        BOOL2BOOL_14 : BOOL2BOOL;
        BOOL2BOOL_17 : BOOL2BOOL;
        UINT2UINT_8 : UINT2UINT;
        E_R_TRIG_5 : E_R_TRIG;
        BOOL2BOOL_21 : BOOL2BOOL;
      END_FBS
      SUBAPPS
        OPC_PUB_EX_5 : OPC_PUB_EX_1(QI := 1, prefix := "FIO_Q_", var1 := "sorter_3_belt", server := WSTRING#"localhost:4840");
        OPC_SUB_EX_6 : OPC_SUB_EX_1(QI := 1, prefix := "CON_", var1 := "sorter_3", server := WSTRING#"localhost:4840");
        OPC_PUB_EX_6 : OPC_PUB_EX_1(QI := 1, prefix := "FIO_Q_", var1 := "sorter_3_turn", server := WSTRING#"localhost:4840");
        SorterLogic_1 : SorterLogic(PackageNum := UINT#3);
        OPC_SUB_EX_9 : OPC_SUB_EX_1(QI := 1, prefix := "FIO_I_", var1 := "at_exit", server := WSTRING#"localhost:4840");
        OPC_PUB_EX_9 : OPC_PUB_EX_1(QI := 1, prefix := "CON_", var1 := "C3", server := WSTRING#"localhost:4840");
        OPC_SUB_EX_3 : OPC_SUB_EX_1(QI := 1, prefix := "FIO_I_", var1 := "reset", server := WSTRING#"localhost:4840");
      END_SUBAPPS
      EVENT_CONNECTIONS
        OPC_SUB_EX_6.INITO TO OPC_PUB_EX_5.INIT;
        START.COLD TO OPC_SUB_EX_6.INIT;
        OPC_PUB_EX_5.INITO TO OPC_PUB_EX_6.INIT;
        OPC_SUB_EX_6.IND TO UINT2UINT_4.REQ;
        UINT2UINT_4.CNF TO SorterLogic_1.IND;
        SorterLogic_1.CNF TO BOOL2BOOL_14.REQ;
        BOOL2BOOL_14.CNF TO OPC_PUB_EX_5.REQ;
        BOOL2BOOL_14.CNF TO OPC_PUB_EX_6.REQ;
        OPC_SUB_EX_6.INITO TO OPC_SUB_EX_9.INIT;
        OPC_SUB_EX_9.IND TO BOOL2BOOL_17.REQ;
        BOOL2BOOL_17.CNF TO SorterLogic_1.C;
        SorterLogic_1.CNT TO UINT2UINT_8.REQ;
        OPC_PUB_EX_6.CNF TO OPC_PUB_EX_9.INIT;
        UINT2UINT_8.CNF TO OPC_PUB_EX_9.REQ;
        E_R_TRIG_5.EO TO SorterLogic_1.ResetC;
        BOOL2BOOL_21.CNF TO E_R_TRIG_5.EI;
        OPC_SUB_EX_9.INITO TO OPC_SUB_EX_3.INIT;
        OPC_SUB_EX_3.IND TO BOOL2BOOL_21.REQ;
      END_CONNECTIONS
      DATA_CONNECTIONS
        OPC_SUB_EX_6.value TO UINT2UINT_4.IN;
        UINT2UINT_4.OUT TO SorterLogic_1.value;
        SorterLogic_1.OUT TO BOOL2BOOL_14.IN;
        BOOL2BOOL_14.OUT TO OPC_PUB_EX_5.value;
        BOOL2BOOL_14.OUT TO OPC_PUB_EX_6.value;
        OPC_SUB_EX_9.value TO BOOL2BOOL_17.IN;
        BOOL2BOOL_17.OUT TO SorterLogic_1.AtExit;
        SorterLogic_1.CV TO UINT2UINT_8.IN;
        UINT2UINT_8.OUT TO OPC_PUB_EX_9.value;
        BOOL2BOOL_21.OUT TO E_R_TRIG_5.QI;
        OPC_SUB_EX_3.value TO BOOL2BOOL_21.IN;
      END_CONNECTIONS
    END_RESOURCE
  END_DEVICE
  MAPPINGS
    Sorting_Station.FIO ON PLC.CPU1.FIO;
    Sorting_Station.E_R_TRIG ON PLC.CPU1.E_R_TRIG;
    Sorting_Station.BOOL2BOOL ON PLC.CPU1.BOOL2BOOL;
    Sorting_Station.BOOL2BOOL_1 ON PLC.CPU1.BOOL2BOOL_1;
    Sorting_Station.UPC_PUB_FIO ON PLC.CPU1.UPC_PUB_FIO;
    Sorting_Station.Start_Light ON PLC.CPU1.Start_Light;
    Sorting_Station.Reset_Light ON PLC.CPU1.Reset_Light;
    Sorting_Station.Stop_Light ON PLC.CPU1.Stop_Light;
    Sorting_Station.ENTRY_CONVEYOR ON PLC.CPU1.ENTRY_CONVEYOR;
    Sorting_Station.EXIT_CONVEYOR ON PLC.CPU1.EXIT_CONVEYOR;
    Sorting_Station.At_Exit ON PLC.CPU1.At_Exit;
    Sorting_Station.Vison_Sensor ON PLC.CPU1.Vison_Sensor;
    Sorting_Station.Stop ON PLC.CPU1.Stop;
    Sorting_Station.Reset ON PLC.CPU1.Reset;
    Sorting_Station.Emergency_Stop ON PLC.CPU1.Emergency_Stop;
    Sorting_Station.Auto ON PLC.CPU1.Auto;
    Sorting_Station.Manual ON PLC.CPU1.Manual;
    Sorting_Station.BOOL2BOOL_2 ON PLC.CPU1.BOOL2BOOL_2;
    Sorting_Station.BOOL2BOOL_3 ON PLC.CPU1.BOOL2BOOL_3;
    Sorting_Station.BOOL2BOOL_4 ON PLC.CPU1.BOOL2BOOL_4;
    Sorting_Station.BOOL2BOOL_5 ON PLC.CPU1.BOOL2BOOL_5;
    Sorting_Station.BOOL2BOOL_6 ON PLC.CPU1.BOOL2BOOL_6;
    Sorting_Station.BOOL2BOOL_7 ON PLC.CPU1.BOOL2BOOL_7;
    Sorting_Station.BOOL2BOOL_8 ON PLC.CPU1.BOOL2BOOL_8;
    Sorting_Station.BOOL2BOOL_9 ON PLC.CPU1.BOOL2BOOL_9;
    Sorting_Station.BOOL2BOOL_10 ON PLC.CPU1.BOOL2BOOL_10;
    Sorting_Station.BOOL2BOOL_11 ON PLC.CPU1.BOOL2BOOL_11;
    Sorting_Station.Start ON PLC.CPU1.Start;
    Sorting_Station.STOP_BLADE ON PLC.CPU1.STOP_BLADE;
    Sorting_Station.BOOL2BOOL_18 ON PLC.CPU1.BOOL2BOOL_18;
    Sorting_Station.E_R_TRIG_2 ON PLC.CPU1.E_R_TRIG_2;
    Sorting_Station.Is_running ON PLC.CPU1.Is_running;
    Sorting_Station.E_F_TRIG ON PLC.CPU1.E_F_TRIG;
    Sorting_Station.Is_running_NOT ON PLC.CPU1.Is_running_NOT;
    Sorting_Station.UINT2UINT ON PLC.CPU1.UINT2UINT;
    Sorting_Station.E_R_TRIG_1 ON PLC.CPU1.E_R_TRIG_1;
    Sorting_Station.Sorter_1 ON PLC.CPU1.Sorter_1;
    Sorting_Station.Sorter_2 ON PLC.CPU1.Sorter_2;
    Sorting_Station.Sorter_3 ON PLC.CPU1.Sorter_3;
    Sorting_Station.OPC_PUB_1_FixID ON PLC.CPU1.OPC_PUB_1_FixID;
    Sorting_Station.OPC_PUB_EX_1 ON SorterUnit1.EMB_RES.OPC_PUB_EX_1;
    Sorting_Station.OPC_PUB_EX_2 ON SorterUnit1.EMB_RES.OPC_PUB_EX_2;
    Sorting_Station.OPC_SUB_EX_4 ON SorterUnit1.EMB_RES.OPC_SUB_EX_4;
    Sorting_Station.OPC_SUB_EX_5 ON SorterUnit2.EMB_RES.OPC_SUB_EX_5;
    Sorting_Station.OPC_PUB_EX_3 ON SorterUnit2.EMB_RES.OPC_PUB_EX_3;
    Sorting_Station.OPC_PUB_EX_4 ON SorterUnit2.EMB_RES.OPC_PUB_EX_4;
    Sorting_Station.OPC_PUB_EX_5 ON SorterUnit3.EMB_RES.OPC_PUB_EX_5;
    Sorting_Station.OPC_SUB_EX_6 ON SorterUnit3.EMB_RES.OPC_SUB_EX_6;
    Sorting_Station.OPC_PUB_EX_6 ON SorterUnit3.EMB_RES.OPC_PUB_EX_6;
    Sorting_Station.OPC_PUB_1_FixID_1 ON PLC.CPU1.OPC_PUB_1_FixID_1;
    Sorting_Station.OPC_PUB_1_FixID_2 ON PLC.CPU1.OPC_PUB_1_FixID_2;
    Sorting_Station.F_SEL ON PLC.CPU1.F_SEL;
    Sorting_Station.UINT2UINT_1 ON PLC.CPU1.UINT2UINT_1;
    Sorting_Station.SorterLogic ON SorterUnit1.EMB_RES.SorterLogic;
    Sorting_Station.UINT2UINT_2 ON SorterUnit1.EMB_RES.UINT2UINT_2;
    Sorting_Station.BOOL2BOOL_12 ON SorterUnit1.EMB_RES.BOOL2BOOL_12;
    Sorting_Station.UINT2UINT_3 ON SorterUnit2.EMB_RES.UINT2UINT_3;
    Sorting_Station.SorterLogic_3 ON SorterUnit2.EMB_RES.SorterLogic_3;
    Sorting_Station.BOOL2BOOL_13 ON SorterUnit2.EMB_RES.BOOL2BOOL_13;
    Sorting_Station.UINT2UINT_4 ON SorterUnit3.EMB_RES.UINT2UINT_4;
    Sorting_Station.SorterLogic_1 ON SorterUnit3.EMB_RES.SorterLogic_1;
    Sorting_Station.BOOL2BOOL_14 ON SorterUnit3.EMB_RES.BOOL2BOOL_14;
    Sorting_Station.OPC_SUB_EX_7 ON SorterUnit1.EMB_RES.OPC_SUB_EX_7;
    Sorting_Station.OPC_SUB_1_FixID ON PLC.CPU1.OPC_SUB_1_FixID;
    Sorting_Station.OPC_PUB_EX_7 ON SorterUnit1.EMB_RES.OPC_PUB_EX_7;
    Sorting_Station.BOOL2BOOL_15 ON SorterUnit1.EMB_RES.BOOL2BOOL_15;
    Sorting_Station.UINT2UINT_5 ON SorterUnit1.EMB_RES.UINT2UINT_5;
    Sorting_Station.UINT2UINT_6 ON PLC.CPU1.UINT2UINT_6;
    Sorting_Station.OPC_SUB_EX_8 ON SorterUnit2.EMB_RES.OPC_SUB_EX_8;
    Sorting_Station.BOOL2BOOL_16 ON SorterUnit2.EMB_RES.BOOL2BOOL_16;
    Sorting_Station.OPC_SUB_EX_9 ON SorterUnit3.EMB_RES.OPC_SUB_EX_9;
    Sorting_Station.BOOL2BOOL_17 ON SorterUnit3.EMB_RES.BOOL2BOOL_17;
    Sorting_Station.UINT2UINT_7 ON SorterUnit2.EMB_RES.UINT2UINT_7;
    Sorting_Station.OPC_PUB_EX_8 ON SorterUnit2.EMB_RES.OPC_PUB_EX_8;
    Sorting_Station.UINT2UINT_8 ON SorterUnit3.EMB_RES.UINT2UINT_8;
    Sorting_Station.OPC_PUB_EX_9 ON SorterUnit3.EMB_RES.OPC_PUB_EX_9;
    Sorting_Station.OPC_SUB_1_FixID_1 ON PLC.CPU1.OPC_SUB_1_FixID_1;
    Sorting_Station.UINT2UINT_9 ON PLC.CPU1.UINT2UINT_9;
    Sorting_Station.OPC_SUB_1_FixID_2 ON PLC.CPU1.OPC_SUB_1_FixID_2;
    Sorting_Station.UINT2UINT_10 ON PLC.CPU1.UINT2UINT_10;
    Sorting_Station.BOOL2BOOL_19 ON SorterUnit1.EMB_RES.BOOL2BOOL_19;
    Sorting_Station.E_R_TRIG_3 ON SorterUnit1.EMB_RES.E_R_TRIG_3;
    Sorting_Station.OPC_SUB_EX_1 ON SorterUnit1.EMB_RES.OPC_SUB_EX_1;
    Sorting_Station.E_R_TRIG_5 ON SorterUnit3.EMB_RES.E_R_TRIG_5;
    Sorting_Station.BOOL2BOOL_21 ON SorterUnit3.EMB_RES.BOOL2BOOL_21;
    Sorting_Station.OPC_SUB_EX_3 ON SorterUnit3.EMB_RES.OPC_SUB_EX_3;
    Sorting_Station.OPC_SUB_EX_2 ON SorterUnit2.EMB_RES.OPC_SUB_EX_2;
    Sorting_Station.E_R_TRIG_4 ON SorterUnit2.EMB_RES.E_R_TRIG_4;
    Sorting_Station.BOOL2BOOL_20 ON SorterUnit2.EMB_RES.BOOL2BOOL_20;
  END_MAPPINGS
END_SYSTEM
